// TIA Portal project "inz_dmuch" (V16)

(* hardware
DEVICE "S7-1200 station_1"  S7-1200 Station
   slot 0: "Rack_0"  S7-1200 Rack  Rack  V1.0
   slot 1: "PLC_1"  CPU 1215C AC/DC/Rly  6ES7 215-1BG40-0XB0  V4.4
*)

// ===== PLC "PLC_1"  CPU 1215C AC/DC/Rly =====

VAR_GLOBAL   // PLC tag table "Default tag table"
   "Clock_Byte" AT %MB0 : Byte;
   "Clock_10Hz" AT %M0.0 : Bool;
   "Clock_5Hz" AT %M0.1 : Bool;
   "Clock_2.5Hz" AT %M0.2 : Bool;
   "Clock_2Hz" AT %M0.3 : Bool;
   "Clock_1.25Hz" AT %M0.4 : Bool;
   "Clock_1Hz" AT %M0.5 : Bool;
   "Clock_0.625Hz" AT %M0.6 : Bool;
   "Clock_0.5Hz" AT %M0.7 : Bool;
   "AI_zasilacz" AT %IW64 : Word;
   "AQ_falownik" AT %QW64 : Word;
   "Norm_cisnienie" AT %MD30 : Real;
   "Scale_cisnienie" AT %MD34 : Real;
   "rozn_cisnien" AT %MD38 : Real;
   "pierwiastek_roznica" AT %MD20 : Real;
   "przeplyw_powietrza" AT %MD24 : Real;
   "wartosc_zadana" AT %MD46 : Real;
   "tryb_pracy" AT %MW54 : Int;
   "kod_bledu" AT %MD50 : DWord;
   "blad" AT %M1.0 : Bool;
   "scaled_input" AT %MD60 : Real;
   "real_output" AT %MD64 : Real;
END_VAR

DATA_BLOCK "Data_Simulation"   // DB2
{ S7_Optimized_Access := 'TRUE' }
VERSION : 0.1
   VAR
      BoolArray : Array[0..5] of Bool;
      Structure : Struct
         MyInt : Int := 2;
         MyReal : Real := 15.2;
         MyBool : Bool;
      END_STRUCT;
   END_VAR
BEGIN
   BoolArray[0] := True;
   BoolArray[3] := True;
END_DATA_BLOCK

ORGANIZATION_BLOCK "Main"   // OB1, LAD, ProgramCycle
TITLE = "Main Program Sweep (Cycle)"
{ S7_Optimized_Access := 'TRUE' }
VERSION : 0.1
   VAR_INPUT
      Initial_Call : Bool;   // Initial call of this OB
      Remanence : Bool;   // =True, if remanent data are available
   END_VAR
BEGIN

REGION Network 1
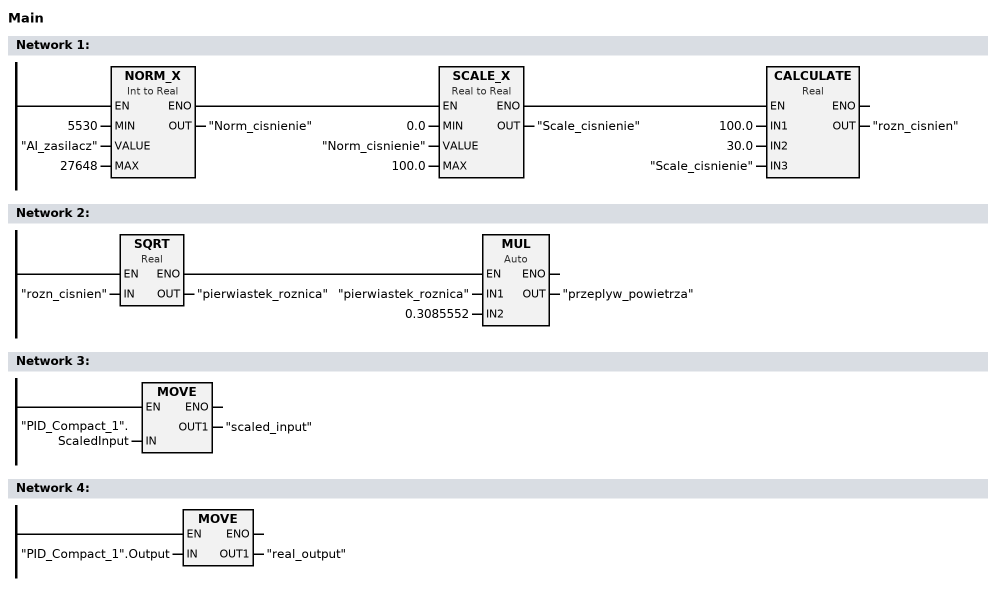
   RUNG wire#powerrail
      { S7_Templates := "[SrcType := Int, DestType := Real]" } Normalize(min := 5530, value := "AI_zasilacz", max := 27648, out => "Norm_cisnienie")
      { S7_Templates := "[SrcType := Real, DestType := Real]" } Scale(min := 0.0, value := "Norm_cisnienie", max := 100.0, out => "Scale_cisnienie")
      { S7_Templates := "SrcType := Real"; S7_Expression := "(IN3*IN2)/IN1" } Calculate(in1 := 100.0, in2 := 30.0, in3 := "Scale_cisnienie", out => "rozn_cisnien")
   END_RUNG
   // the same network as SCL:
   "Norm_cisnienie" := NORM_X(MIN := 5530, VALUE := "AI_zasilacz", MAX := 27648);
   "Scale_cisnienie" := SCALE_X(MIN := 0.0, VALUE := "Norm_cisnienie", MAX := 100.0);
   "rozn_cisnien" := ("Scale_cisnienie"*30.0)/100.0;
END_REGION

REGION Network 2
   "pierwiastek_roznica" := SQRT("rozn_cisnien");
   "przeplyw_powietrza" := "pierwiastek_roznica" * 0.3085552;
END_REGION

REGION Network 3
   RUNG wire#powerrail
      Move(in := "PID_Compact_1".ScaledInput, out1 => "scaled_input")
   END_RUNG
   // the same network as SCL:
   "scaled_input" := "PID_Compact_1".ScaledInput;
END_REGION

REGION Network 4
   RUNG wire#powerrail
      Move(in := "PID_Compact_1".Output, out1 => "real_output")
   END_RUNG
   // the same network as SCL:
   "real_output" := "PID_Compact_1".Output;
END_REGION
END_ORGANIZATION_BLOCK

ORGANIZATION_BLOCK "Cyclic interrupt"   // OB30, LAD, CyclicInterrupt
TITLE = pid
{ S7_Optimized_Access := 'TRUE' }
VERSION : 0.1
   VAR_INPUT
      Initial_Call : Bool;   // Initial call of this OB
      Event_Count : Int;   // Events discarded
   END_VAR
BEGIN

REGION Network 1
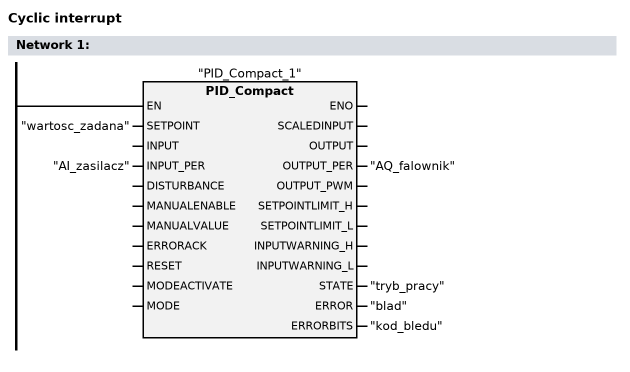
   "PID_Compact_1"(Setpoint := "wartosc_zadana",   // PID_Compact
                   Input_PER := "AI_zasilacz",
                   Output_PER => "AQ_falownik",
                   State => "tryb_pracy",
                   Error => "blad",
                   ErrorBits => "kod_bledu");
END_REGION
END_ORGANIZATION_BLOCK